# EPICS autosave request: measCompApp/Db/measCompAnalogOut_settings.req
$(P)$(R)Pulse
$(P)$(R)TweakVal
$(P)$(R).DRVL
$(P)$(R).DRVH
